FUNCTION_BLOCK FB_OM_Config
VAR_INPUT
END_VAR
VAR_OUTPUT
	eCurrentState : E_MachineState := E_MachineState.MACHINESTATE_Idle;
END_VAR
VAR
	bFirstCycle				: BOOL := TRUE;
	stError					: ST_Error;
	bError					: BOOL;
	bBusy					: BOOL;
	
	//ConfigActions
	nStateA_ConfigAction	: USINT;
	bActivate				: BOOL;
	nActivateCnt1			: USINT; //allg Zählvariable
	
	bSaveCurrConfig			: BOOL;
	bLoadConfig				: BOOL;
	bDeleteConfig			: BOOL;
	
	nStateA_CheckObjProps	: USINT;
	iter					: FB_ObjCollectIteratorDeep;
	pObject					: POINTER TO FB_Object;
	nCheckObjCounter		: USINT;
	
	nStateA_Reset			: USINT;
	i						: UINT;
	bSetupDefaultObjOk		: BOOL;
	timer					: TON;
	
	bWriteXYAxisPara		: BOOL;
	nStateA_WriteXYAxisPara	: USINT;
	
	bSimError				: BOOL;
END_VAR

IF bFirstCycle THEN
	bFirstCycle := FALSE;
	bLoadConfig := fbConfiguration.P_bConfigSaved;
	eCurrentState := E_MachineState.MACHINESTATE_Active;	
END_IF

IF eCurrentState = E_MachineState.MACHINESTATE_Active THEN
	IF bLoadConfig THEN
		fbConfiguration.A_Load(bExecute:= TRUE);
		IF NOT fbConfiguration.bBusy THEN
			IF fbConfiguration.bError THEN
				bError := TRUE;
				fbErrorList.M_Add(stError);
			ELSE
				bActivate := TRUE;
			END_IF
			fbConfiguration.A_Load(bExecute:= FALSE);
			bLoadConfig := FALSE;
			//bei erfolg Konfiguration laden
		END_IF
	ELSIF bDeleteConfig THEN
		fbConfiguration.A_Delete(bExecute:= TRUE);
		IF NOT fbConfiguration.bBusy THEN
			IF fbConfiguration.bError THEN
				bError := TRUE;
				fbErrorList.M_Add(stError);
			END_IF
			fbConfiguration.A_Delete(bExecute:= FALSE);
			bDeleteConfig := FALSE;
		END_IF
	ELSIF bActivate THEN	//Konfiguration aktivieren
		fbConfiguration.A_Activate(bExecute:= TRUE);
		IF NOT fbConfiguration.bBusy THEN
			IF fbConfiguration.bError THEN
				bError := TRUE;
				fbErrorList.M_Add(fbConfiguration.stError);
			END_IF
			fbConfiguration.A_Activate(bExecute:= FALSE);
			bActivate := FALSE;
		END_IF
	ELSIF bSaveCurrConfig THEN
		fbConfiguration.A_Save(bExecute:= TRUE);
		IF NOT fbConfiguration.bBusy THEN
			IF fbConfiguration.bError THEN
				bError := TRUE;
				fbErrorList.M_Add(stError);
			END_IF
			fbConfiguration.A_Save(bExecute:= FALSE);
			bSaveCurrConfig := FALSE;
		END_IF
	END_IF

	IF NOT (bActivate OR bSaveCurrConfig OR bLoadConfig OR bDeleteConfig) THEN
		IF bError THEN
			eCurrentState := E_MachineState.MACHINESTATE_Error;
		ELSE
			eCurrentState := E_MachineState.MACHINESTATE_Idle;
		END_IF
	END_IF
	
ELSIF eCurrentState = E_MachineState.MACHINESTATE_Reset THEN
	A_Reset();
	IF nStateA_Reset = 80 THEN
		nStateA_Reset := 0;
		bError := FALSE;
		eCurrentState := E_MachineState.MACHINESTATE_Idle;
	ELSIF nStateA_Reset = 99 THEN
		nStateA_Reset := 0;
		eCurrentState := E_MachineState.MACHINESTATE_Error;
	END_IF
ELSIF eCurrentState = E_MachineState.MACHINESTATE_Idle THEN
	//Auf Fehler der Hardware reagieren
	IF PerformHardware.bError THEN
		eCurrentState := E_MachineState.MACHINESTATE_Error;
	END_IF
END_IF

IF bSimError THEN
	eCurrentState := E_MachineState.MACHINESTATE_Error;
END_IF

METHOD M_Delete : ERRORID
VAR_INPUT
END_VAR
IF eCurrentState = E_MachineState.MACHINESTATE_Idle THEN
	bDeleteConfig := TRUE;
	eCurrentState := E_MachineState.MACHINESTATE_Active;
END_IF
END_METHOD

METHOD M_Activate : ERRORID
VAR_INPUT
END_VAR
IF eCurrentState = E_MachineState.MACHINESTATE_Idle THEN
	bActivate := TRUE;
	eCurrentState := E_MachineState.MACHINESTATE_Active;
ELSE
	M_Activate := E_ErrorIdCmd.ERRORID_InvalidState;
END_IF
END_METHOD

METHOD M_ResetError
VAR_INPUT
END_VAR
IF eCurrentState = E_MachineState.MACHINESTATE_Error THEN
	eCurrentState := E_MachineState.MACHINESTATE_Reset;
	bError := FALSE;
END_IF
END_METHOD

METHOD M_Save : ERRORID
VAR_INPUT
END_VAR
IF eCurrentState = E_MachineState.MACHINESTATE_Idle THEN
	bSaveCurrConfig := TRUE;
	eCurrentState := E_MachineState.MACHINESTATE_Active;
ELSE
	M_Save := E_ErrorIdCmd.ERRORID_InvalidState;
END_IF
END_METHOD

ACTION A_Reset:
//In Config gehen die Objekte selber nicht in Error, da an diesen keine Actions ausgeführt werden
//Es kann also nur die Hardware in Error gehen, folglich braucht auch nur dieses zurückgesetzt werden
IF nStateA_Reset = 0 THEN
	IF PerformHardware.bError THEN
		PerformHardware.A_ResetError();
		timer(IN:= TRUE, PT:=T#20S);
		IF timer.Q THEN
			timer(IN:= FALSE);
			nStateA_Reset := 99;
		END_IF
	ELSE
		timer(IN:= FALSE);
		nStateA_Reset := 80;
	END_IF	
END_IF
END_ACTION

ACTION A_CheckObjProps:
IF nStateA_CheckObjProps = 0 THEN
	nCheckObjCounter := 0;
	fbObjectDirectory.P_pDeviceCollection^.M_GetIterator(iter);
	nStateA_CheckObjProps := 1;
END_IF

WHILE iter.pNode > 0 AND_THEN iter.pNode^.P_pObject > 0 DO
	pObject := iter.pNode^.P_pObject;
	nCheckObjCounter := nCheckObjCounter + 1;
	stError.ObjectId := pObject^.P_nObjectID;
	stError.ErrorId := pObject^.M_CheckProps();
	IF stError.ErrorId > 0 THEN
		nStateA_CheckObjProps := 99;
		RETURN;
	END_IF
	iter.M_Increment();
	IF nCheckObjCounter = 100 THEN
		nCheckObjCounter := 0;
		RETURN;
	END_IF
END_WHILE

nStateA_CheckObjProps := 80;
END_ACTION

END_FUNCTION_BLOCK

(* stored: Version 1.1.0.1, ProductVersion 3.1.4020.12
   POU FB_OM_Config: Id {13324866-91bb-4b1a-9632-ffce285e2634}, SpecialFunc None
   Method M_Delete: Id {6ab821d4-d9c0-4ba0-b1bc-ae3d2e77db61}
   Method M_Activate: Id {6ec696c5-e2eb-4087-90b6-079772f2791b}
   Method M_ResetError: Id {8f9c9332-5f48-4251-bd01-133545991371}
   Method M_Save: Id {a15da87b-9ca7-4863-bbb7-5177b1c55f85}
   Action A_Reset: Id {be0b7177-997a-4af4-bd21-a1c5e13406f4}
   Action A_CheckObjProps: Id {fdef220d-830e-41e0-938c-3c6061f2fe0f} *)
